// TwinCAT 3 PLC project MicroTestStandREF
// ProgramVersion: 3.1.4020.5
// libraries:
//   lcls-twincat-motion, * (SLAC)
//   lcls2-cc-lib, * (SLAC)
//   Tc2_Standard, * (Beckhoff Automation GmbH)
//   Tc2_System, * (Beckhoff Automation GmbH)
//   Tc2_Utilities, * (Beckhoff Automation GmbH)
//   Tc3_Module, * (Beckhoff Automation GmbH)
//   VisuDialogs
//   VisuSymbols,3.5.10.0,System
// project tree:
//   DUTs/ DUT_MotionStage_Extras.TcDUT
//   / GlobalTextList.TcGTLO, PlcTask.TcTTO (not stored), VISU_TASK.TcTTO (not stored)
//   POUs/ Main.TcPOU
//   VISUs/ Visualization.TcVIS, VisualizationManager.TcVMO (not stored), VISU_MotionStage.TcVIS
// real-time tasks:
//   TASK PlcTask: cycle T#1ms, priority 20, ADS port 350
//   TASK VISU_TASK: cycle T#200000us, priority 30, ADS port 351
// motion (NC):
//   TASK NC-Task 1 SAF: cycle T#1ms, priority 4, ADS port 501
//   TASK NC-Task 1 SVB: cycle T#1ms, priority 8, ADS port 511
//   AXIS MMS_Y (id 1)
//     Dynamic: AccelerationMaximum=200, DecelerationMaximum=200, Acceleration=200, Deceleration=200, Jerk=500, DelayTime=0.004
//     Velo: Maximum=65
//     TargetPosControl: Range=0.002, Time=0.25
//     OtherSettings: AllowMotionCmdToSlave=true
//     encoder EncType=29
//       EncPara: ScaleFactorNumerator=5e-05, Offset=-214686.941, MaxCount=#xffffffff, ReferenceSystem=1
//         Inc: RefSoftSyncMask=#x0000ffff
//     drive DrvType=24
//       Analog: VeloReferenz=100, ScaleFactorActTorque=0.1
//       TimeComp: TaskDelayCycles=1
//     controller CtrType=2
//       CtrPara: PriorControlFactor=1
//         PosDiffControl: Range=1
//         PID: PosKp=20, PosExtKp=1, PosExtVelo=0.1, DeadBandPosition=0.002
//         Observer: BandWidth=20
// I/O:
//   DEVICE Device 1 (EtherCAT), AmsNetId 172.21.148.185.2.1
//     EK1200 [EK1200-5000 EtherCAT Power supply (2A E-Bus)]
//       EL6695 [EL6695 EtherCAT Bridge terminal (Primary)]
//       EK1110 [EK1110 EtherCAT extension]
//     EK1100 [EK1100 EtherCAT Coupler (2A E-Bus)]
//       EL7041 [EL7041 1Ch. Stepper motor output stage (50V, 5A)]
//       EL5042 [EL5042 2Ch. BiSS-C Encoder]
//       EL2004 [EL2004 4Ch. Dig. Output 24V, 0.5A]
//       EL3314 [EL3314 4Ch. Ana. Input Thermocouple (TC)]
//       EL3052 [EL3052 2Ch. Ana. Input 4-20mA]
//       EL3062 [EL3062 2Ch. Ana. Input 0-10V]
//       EL4004 [EL4004 4Ch. Ana. Output 0-10V, 12bit]
//       EL9011 [EL9011 End Terminal]
// variable links:
//   (this object) <-> Device 1 (EtherCAT)/EK1100/EL5042
//     Enc/Inputs/In/nComState @bit 1 <-> WcState/InputToggle
//     Enc/Inputs/In/nComState <-> WcState/WcState
//     Enc/Inputs/In/nDataIn1 <-> FB Inputs Channel 1/Position
//     Enc/Inputs/In/nState1 @bit 12 <-> FB Inputs Channel 1/Status/Diag
//     Enc/Inputs/In/nState1 @bit 1 <-> FB Inputs Channel 1/Status/Error
//     Enc/Inputs/In/nState1 @bit 14 <-> FB Inputs Channel 1/Status/Input cycle counter
//     Enc/Inputs/In/nState1 @bit 2 <-> FB Inputs Channel 1/Status/Ready
//     Enc/Inputs/In/nState1 @bit 13 <-> FB Inputs Channel 1/Status/TxPDO State
//     Enc/Inputs/In/nState1 <-> FB Inputs Channel 1/Status/Warning
//   (this object) <-> Device 1 (EtherCAT)/EK1100/EL7041
//     Drive/Inputs/In/nState1 @bit 3 <-> STM Status/Status/Error
//     Drive/Inputs/In/nState1 @bit 5 <-> STM Status/Status/Moving negative
//     Drive/Inputs/In/nState1 @bit 4 <-> STM Status/Status/Moving positive
//     Drive/Inputs/In/nState1 @bit 1 <-> STM Status/Status/Ready
//     Drive/Inputs/In/nState1 <-> STM Status/Status/Ready to enable
//     Drive/Inputs/In/nState1 @bit 6 <-> STM Status/Status/Torque reduced
//     Drive/Inputs/In/nState1 @bit 2 <-> STM Status/Status/Warning
//     Drive/Inputs/In/nState2 @bit 5 <-> STM Status/Status/Sync error
//     Drive/Inputs/In/nState2 @bit 7 <-> STM Status/Status/TxPDO Toggle
//     Drive/Inputs/In/nState4 @bit 1 <-> WcState/InputToggle
//     Drive/Inputs/In/nState4 <-> WcState/WcState
//     Drive/Outputs/Out/nCtrl1 <-> STM Control/Control/Enable
//     Drive/Outputs/Out/nCtrl1 @bit 2 <-> STM Control/Control/Reduce torque
//     Drive/Outputs/Out/nCtrl1 @bit 1 <-> STM Control/Control/Reset
//     Drive/Outputs/Out/nDataOut2[0] <-> STM Velocity/Velocity
//   MicroTestStandPPM Instance <-> Device 1 (EtherCAT)/EK1100/EL2004
//     PlcTask Outputs/Main.M1.bBrakeRelease <-> Channel 1/Output
//     PlcTask Outputs/Main.fbPPM.fbGige.bGigePower <-> Channel 2/Output
//   MicroTestStandPPM Instance <-> Device 1 (EtherCAT)/EK1100/EL3062
//     PlcTask Inputs/Main.fbPPM.fbPowerMeter.iVoltageINT <-> AI Standard Channel 1/Value
//   MicroTestStandPPM Instance <-> Device 1 (EtherCAT)/EK1100/EL3314
//     PlcTask Inputs/Main.fbPPM.fbPowerMeter.fbThermoCouple.bError <-> TC Inputs Channel 1/Status/Error
//     PlcTask Inputs/Main.fbPPM.fbPowerMeter.fbThermoCouple.bOverrange <-> TC Inputs Channel 1/Status/Overrange
//     PlcTask Inputs/Main.fbPPM.fbPowerMeter.fbThermoCouple.bUnderrange <-> TC Inputs Channel 1/Status/Underrange
//     PlcTask Inputs/Main.fbPPM.fbPowerMeter.fbThermoCouple.iRaw <-> TC Inputs Channel 1/Value
//     PlcTask Inputs/Main.fbPPM.fbYagThermoCouple.bError <-> TC Inputs Channel 2/Status/Error
//     PlcTask Inputs/Main.fbPPM.fbYagThermoCouple.bOverrange <-> TC Inputs Channel 2/Status/Overrange
//     PlcTask Inputs/Main.fbPPM.fbYagThermoCouple.bUnderrange <-> TC Inputs Channel 2/Status/Underrange
//     PlcTask Inputs/Main.fbPPM.fbYagThermoCouple.iRaw <-> TC Inputs Channel 2/Value
//   MicroTestStandPPM Instance <-> Device 1 (EtherCAT)/EK1100/EL4004
//     PlcTask Outputs/Main.fbPPM.fbGige.iIlluminatorINT <-> AO Outputs Channel 1/Analog output
//   MicroTestStandPPM Instance <-> Device 1 (EtherCAT)/EK1100/EL5042
//     PlcTask Inputs/Main.iRawEncoder <-> FB Inputs Channel 1/Position
//   MicroTestStandPPM Instance <-> Device 1 (EtherCAT)/EK1100/EL7041
//     PlcTask Inputs/Main.M1.bLimitBackwardEnable <-> STM Status/Status/Digital input 2
//     PlcTask Inputs/Main.M1.bLimitForwardEnable <-> STM Status/Status/Digital input 1
//   MicroTestStandPPM Instance <-> NC-Task 1 SAF/Axes/MMS_Y
//     PlcTask Inputs/Main.M1.Axis.NcToPlc <-> Outputs/ToPlc
//     PlcTask Outputs/Main.M1.Axis.PlcToNc <-> Inputs/FromPlc

// ---- DUTs/DUT_MotionStage_Extras.TcDUT
TYPE DUT_MotionStage_Extras :
STRUCT
	fVisuStep: LREAL;
	bVisuLowLim: BOOL;
	bVisuHighLim: BOOL;
END_STRUCT
END_TYPE

// ---- POUs/Main.TcPOU
PROGRAM Main
VAR
	{attribute 'pytmc' := '
        pv: TST:REF:MMS:01
		io: io
	'}
	{attribute 'TcLinkTo' := '.bLimitForwardEnable  := TIIB[EL7041]^STM Status^Status^Digital input 1;
	                          .bLimitBackwardEnable := TIIB[EL7041]^STM Status^Status^Digital input 2;
	                          .bBrakeRelease        := TIIB[EL2004]^Channel 1^Output'}
	M1: DUT_MotionStage;
	M1_Extras: DUT_MotionStage_Extras;
	
	{attribute 'pytmc' := '
		pv: TST:REF
		io: io
	'}
	{attribute 'TcLinkTo' := '.fbLaser.iLaserINT := TIIB[EL4004]^AO Outputs Channel 1^Analog output;
							  .fbLaser.iShutdownINT := TIIB[EL4004]^AO Outputs Channel 2^Analog output'}
	fbREF: FB_REF;
	
	{attribute 'pytmc' := '
		pv: TST:REF:MMS:01:ENC_RAW
		io: i
	'}
	iAdjustedEncoder: UDINT;
	iRawEncoder AT %I*: ULINT;
	iMaxLINT: ULINT := 18446744073709551615;
	
	bLaserPower: BOOL;
	
	bStartup: BOOL := TRUE;
END_VAR

fbREF(stYStage := M1);
M1.bHardwareEnable := TRUE;
iAdjustedEncoder :=  ULINT_TO_UDINT(iMaxLINT - iRawEncoder);

M1_Extras.bVisuHighLim := NOT M1.bAllForwardEnable;
M1_Extras.bVisuLowLim := NOT M1.bAllBackwardEnable;

IF bStartup THEN
	bStartup := FALSE;
	M1.fVelocity := 1;
	M1.fAcceleration := 200;
	M1.fDeceleration := 200;
END_IF

END_PROGRAM

// ---- GlobalTextList.TcGTLO
TEXTLIST GlobalTextList
  593 = '%f'
  964 = '%X'
  957 = '+'
  951 = '-'
  960 = '0 = Default Acceleration'
  962 = '0 = Default Deceleration'
  959 = 'Acceleration: %f'
  504 = 'Cam Power'
  955 = 'Clear'
  582 = 'Close Screen'
  949 = 'Control'
  684 = 'Controls'
  594 = 'Current Position'
  961 = 'Deceleration: %f'
  965 = 'Error Code'
  963 = 'Error:'
  953 = 'GO'
  954 = 'GO to set position'
  595 = 'High Limit Hit Indicator'
  768 = 'Illuminator: %f %'
  479 = 'Laser Power'
  116 = 'Laser Suppress: %f %'
  896 = 'Laser: %f %'
  592 = 'Low Limit Hit Indicator'
  30 = 'Motion Stage'
  460 = 'Motor'
  596 = 'Moving:'
  311 = 'Parker Stage'
  109 = 'PM TC: %f C'
  658 = 'PM Temp: %f C'
  598 = 'Power Meter: %f V'
  921 = 'PPM'
  890 = 'Raw count: %d'
  7 = 'Raw count: %f'
  274 = 'Readbacks'
  333 = 'REF'
  950 = 'Set Position'
  470 = 'Settings'
  591 = 'Status'
  952 = 'Step Size'
  956 = 'STOP'
  958 = 'Velocity: %f'
  316 = 'Yag Temp: %f C'
END_TEXTLIST

// ---- VISUs/Visualization.TcVIS
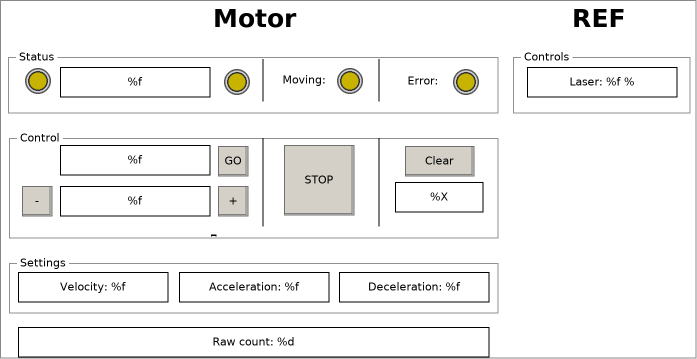
VISUALIZATION Visualization  // 697x359
    Label (14,3 482x30), "Motor"
    Label (503,3 192x30), "REF"
    Rectangle (18,327 471x30), "Raw count: %d", text variable: Main.iAdjustedEncoder
    GroupBox (513,49 177x64), "Controls"
        Rectangle (14,18 150x30), "Laser: %f %", text variable: Main.fbREF.fbLaser.fLaserPercent
            OnMouseDown: write the text variable via Default, min 0, max 100
    Frame (-7,32 520x300)
        shows VISU_MotionStage(VisuMotionStage := Main.M1, Extras := Main.M1_Extras)
END_VISUALIZATION

// ---- VISUs/VISU_MotionStage.TcVIS
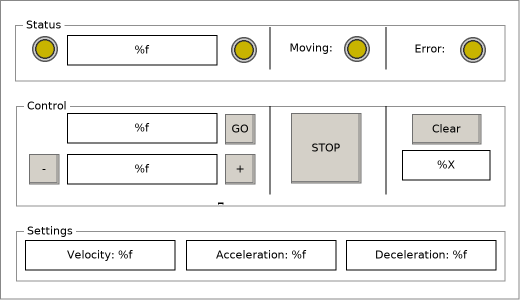
VISUALIZATION VISU_MotionStage  // 520x300
VAR_IN_OUT
	VisuMotionStage: DUT_MotionStage;
	Extras: DUT_MotionStage_Extras;
END_VAR
    GroupBox (15,17 490x64), "Status"
        Lamp1 (15,17 30x30), tooltip "Low Limit Hit Indicator", variable: Extras.bVisuLowLim, style: Lamp-Lamp1-Yellow
        Rectangle (52,18 150x30), "%f", tooltip "Current Position", text variable: VisuMotionStage.stAxisStatus.fActPosition
        Lamp1 (214,18 30x30), tooltip "High Limit Hit Indicator", variable: Extras.bVisuHighLim, style: Lamp-Lamp1-Yellow
        Lamp1 (327,17 30x30), variable: VisuMotionStage.bBusy, style: Lamp-Lamp1-Yellow
        Label (262,16 68x30), "Moving:"
        Line (371,52) (371,10)
        Lamp1 (443,18 30x30), variable: VisuMotionStage.bError, style: Lamp-Lamp1-Yellow
    Rectangle (218,203 5x0)
    GroupBox (16,98 489x108), "Control"
        Rectangle (51,15 150x30), "%f", tooltip "Set Position", text variable: VisuMotionStage.fPosition
            OnMouseDown: write the text variable via Default
        Button (13,56 30x30), "-"
            OnMouseDown: execute {
                VisuMotionStage.nCommand := 3;
                VisuMotionStage.fPosition := VisuMotionStage.stAxisStatus.fActPosition - Extras.fVisuStep;
                VisuMotionStage.bExecute := TRUE;
            }
        Rectangle (51,56 150x30), "%f", tooltip "Step Size", text variable: Extras.fVisuStep
            OnMouseDown: write the text variable via Default
        Button (209,16 30x30), "GO", tooltip "GO to set position"
            OnMouseDown: execute { VisuMotionStage.nCommand := 3; VisuMotionStage.bExecute := TRUE; }
        Line (254,96) (254,8)
        Line (370,96) (370,8)
        Button (396,16 69x30), "Clear"
            tap VisuMotionStage.bReset
        Button (275,15 70x70), "STOP", tooltip "GO to set position"
            OnMouseDown: execute { VisuMotionStage.bExecute := FALSE; }
        Button (209,56 30x30), "+"
            OnMouseDown: execute {
                VisuMotionStage.nCommand := 3;
                VisuMotionStage.fPosition := VisuMotionStage.stAxisStatus.fActPosition + Extras.fVisuStep;
                VisuMotionStage.bExecute := TRUE;
            }
    GroupBox (16,223 489x58), "Settings"
        Rectangle (9,17 150x30), "Velocity: %f", text variable: VisuMotionStage.fVelocity
            OnMouseDown: write the text variable via Default
        Rectangle (170,17 150x30), "Acceleration: %f", tooltip "0 = Default Acceleration", text variable: VisuMotionStage.fAcceleration
            OnMouseDown: write the text variable via Default
        Rectangle (330,17 150x30), "Deceleration: %f", tooltip "0 = Default Deceleration", text variable: VisuMotionStage.fDeceleration
            OnMouseDown: write the text variable via Default
    Line (270,69) (270,27)
    Label (396,34 68x30), "Error:"
    Rectangle (402,150 88x30), "%X", tooltip "Error Code", text variable: VisuMotionStage.stAxisStatus.nErrorId
END_VISUALIZATION
